(* CODESYS project exsamen m6 no scada.project
   CustomField01_name: CustomField01
   CustomField08_name: CustomField08
   CustomField06_name: CustomField06
   Title: ATV_IMC_Template
   CustomField09_name: CustomField09
   CustomField07_name: CustomField07
   CustomField05_name: CustomField05
   CustomField02_name: CustomField02
   Description: This template can be used for a correct interface with the local drive. the MANDATORY_AT_EACH_CYCLE program must be called like it is done in this application.
   CustomField04_name: CustomField04
   CustomField10_name: CustomField10
   Version: 0.0.0.0
   Company: Schneider Electric
   CustomField03_name: CustomField03

Project tree, tasks and I/O mapping:
  MyController : TM241CE24R, Schneider Electric, order no. TM241CE24R, version 4.0.3.8
    application Application
      task MAST (cyclic, interval 20 ms, priority 15, watchdog 100 ms x 1) calls progprinc
      function HiddenPOU [ST]
      global variables GVL
      program progprinc [SFC]: RojoManual, PlataManual, NegraManual, PlataAuto, NegroAuto, RojoAuto
      function block POU [LD]
      visualisation scada
    DI : Digital Inputs, Schneider Electric, version 4.0.3.8
        input  ibDI_IB1 : BYTE  // IB1
        unmapped channels: IW0
    DQ : Digital Outputs, Schneider Electric, version 4.0.3.8
        output qwDQ_QW0 : WORD  // QW0
        output qbDQ_QB1 : BYTE  // QB1
    Counters : Counters, Schneider Electric, version 4.0.3.8
    Pulse_Generators : Pulse Generators, Schneider Electric, version 4.0.3.8
    Cartridge_1 : Cartridge, Schneider Electric, version 4.0.3.8
    IO_Bus : IO bus - TM3, Schneider Electric, version 4.0.3.8
    COM_Bus : COM bus, Schneider Electric, version 4.0.3.8
    Ethernet_1 : Ethernet Network, Schneider Electric, version 4.0.3.8
    Serial_Line_1 : Serial line, Schneider Electric, version 4.0.3.8
      SoMachine_Network_Manager : SoMachine-Network Manager, Schneider Electric, version 4.0.0.2
    Serial_Line_2 : Serial line, Schneider Electric, version 4.0.3.8
      Modbus_Manager : Modbus Manager, Schneider Electric, version 4.0.0.2
  text list GlobalTextList
*)

// MyController/Application/GVL
VAR_GLOBAL
	Marcha: BOOL;
	Confirmar: BOOL;
	Modo: BOOL;
	
	Bot: INT;
	
	SelecPlata: BOOL;
	SensAlmacenPlata: BOOL;
	SensCilPlata: BOOL;
	
	SelecRojo: BOOL;
	SensAlmacenRojo: BOOL;
	SensCilRojo: BOOL;
	
	SelecNegro: BOOL;
	SensAlmacenNego: BOOL;
	SensCilNegro: BOOL;
	

	Cinta: BOOL;
	Seleccion: BOOL;
END_VAR

// MyController/Application/progprinc
PROGRAM progprinc
VAR
	MarchaPanel: BOOL;
	etapa_0: BOOL;
	etapa_1: BOOL;
	FuncManRojo: POU;
	piezasrojas: INT;
	piezasnegras: INT;
	piezasplata: INT;
	FunManNegra: POU;
	FuncManPlata: POU;
	FuncAutoPlata: POU;
	FuncAutoNegra: POU;
	FuncAutoRoja: POU;

END_VAR

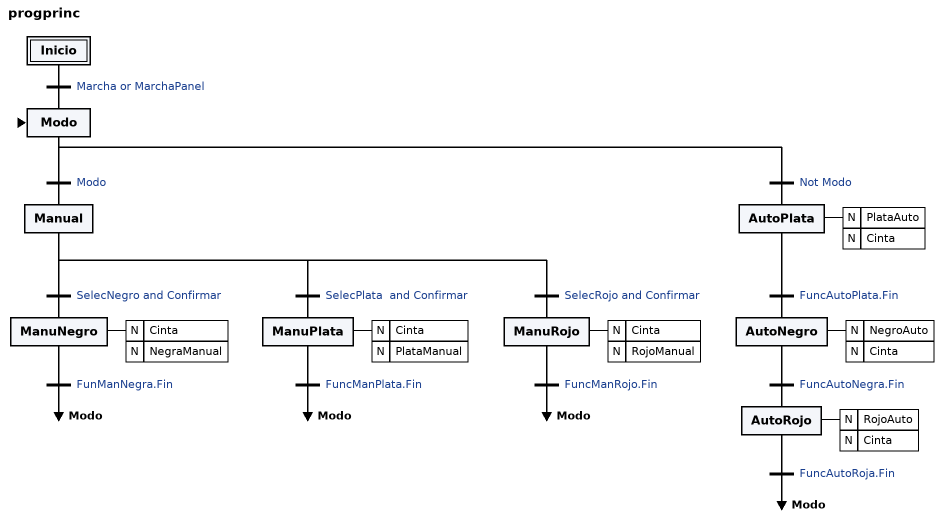
INITIAL_STEP Inicio:
END_STEP
TRANSITION FROM Inicio TO Modo
    := Marcha or MarchaPanel;
END_TRANSITION
STEP Modo:
END_STEP
TRANSITION FROM Modo TO Manual
    := Modo;
END_TRANSITION
STEP Manual:
END_STEP
TRANSITION FROM Manual TO ManuNegro
    := SelecNegro and Confirmar;
END_TRANSITION
STEP ManuNegro:
    Cinta(N);
    NegraManual(N);
END_STEP
TRANSITION FROM ManuNegro TO Modo
    := FunManNegra.Fin;
END_TRANSITION
TRANSITION FROM Manual TO ManuPlata
    := SelecPlata and Confirmar;
END_TRANSITION
STEP ManuPlata:
    Cinta(N);
    PlataManual(N);
END_STEP
TRANSITION FROM ManuPlata TO Modo
    := FuncManPlata.Fin;
END_TRANSITION
TRANSITION FROM Manual TO ManuRojo
    := SelecRojo and Confirmar;
END_TRANSITION
STEP ManuRojo:
    Cinta(N);
    RojoManual(N);
END_STEP
TRANSITION FROM ManuRojo TO Modo
    := FuncManRojo.Fin;
END_TRANSITION
TRANSITION FROM Modo TO AutoPlata
    := Not Modo;
END_TRANSITION
STEP AutoPlata:
    PlataAuto(N);
    Cinta(N);
END_STEP
TRANSITION FROM AutoPlata TO AutoNegro
    := FuncAutoPlata.Fin;
END_TRANSITION
STEP AutoNegro:
    NegroAuto(N);
    Cinta(N);
END_STEP
TRANSITION FROM AutoNegro TO AutoRojo
    := FuncAutoNegra.Fin;
END_TRANSITION
STEP AutoRojo:
    RojoAuto(N);
    Cinta(N);
END_STEP
TRANSITION FROM AutoRojo TO Modo
    := FuncAutoRoja.Fin;
END_TRANSITION

ACTION RojoManual:
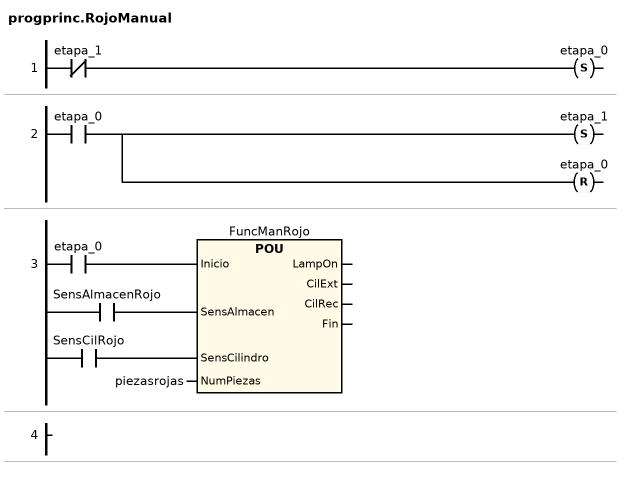
// NETWORK 1
etapa_0 S= NOT etapa_1;

// NETWORK 2
etapa_1 S= etapa_0;
etapa_0 R= etapa_0;

// NETWORK 3
FuncManRojo(
    Inicio := etapa_0,
    SensAlmacen := SensAlmacenRojo,
    SensCilindro := SensCilRojo,
    NumPiezas := piezasrojas); // POU

// NETWORK 4
END_ACTION

ACTION PlataManual:
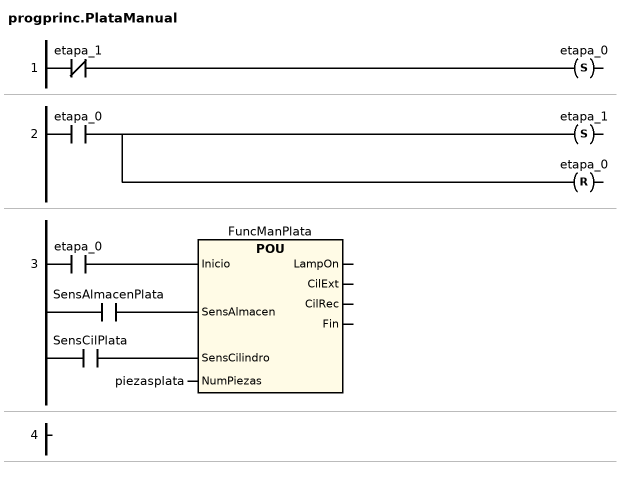
// NETWORK 1
etapa_0 S= NOT etapa_1;

// NETWORK 2
etapa_1 S= etapa_0;
etapa_0 R= etapa_0;

// NETWORK 3
FuncManPlata(
    Inicio := etapa_0,
    SensAlmacen := SensAlmacenPlata,
    SensCilindro := SensCilPlata,
    NumPiezas := piezasplata); // POU

// NETWORK 4
END_ACTION

ACTION NegraManual:
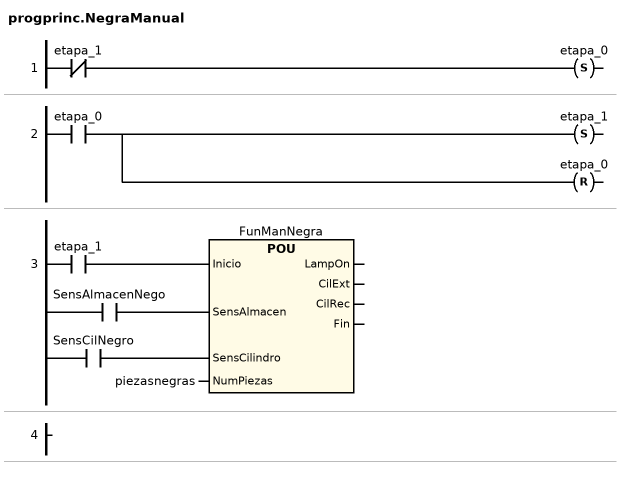
// NETWORK 1
etapa_0 S= NOT etapa_1;

// NETWORK 2
etapa_1 S= etapa_0;
etapa_0 R= etapa_0;

// NETWORK 3
FunManNegra(
    Inicio := etapa_1,
    SensAlmacen := SensAlmacenNego,
    SensCilindro := SensCilNegro,
    NumPiezas := piezasnegras); // POU

// NETWORK 4
END_ACTION

ACTION PlataAuto:
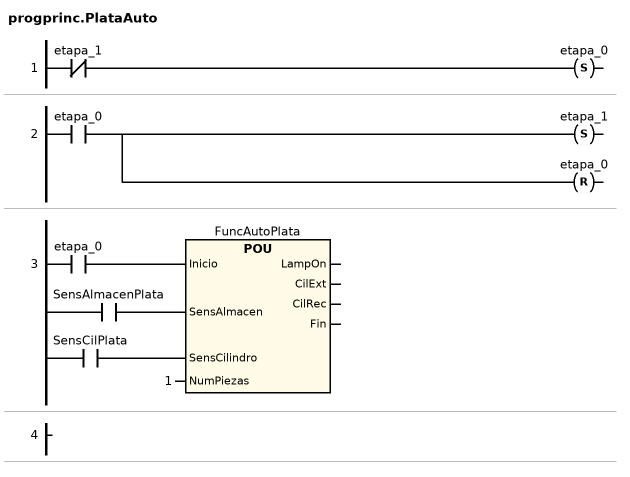
// NETWORK 1
etapa_0 S= NOT etapa_1;

// NETWORK 2
etapa_1 S= etapa_0;
etapa_0 R= etapa_0;

// NETWORK 3
FuncAutoPlata(
    Inicio := etapa_0,
    SensAlmacen := SensAlmacenPlata,
    SensCilindro := SensCilPlata,
    NumPiezas := 1); // POU

// NETWORK 4
END_ACTION

ACTION NegroAuto:
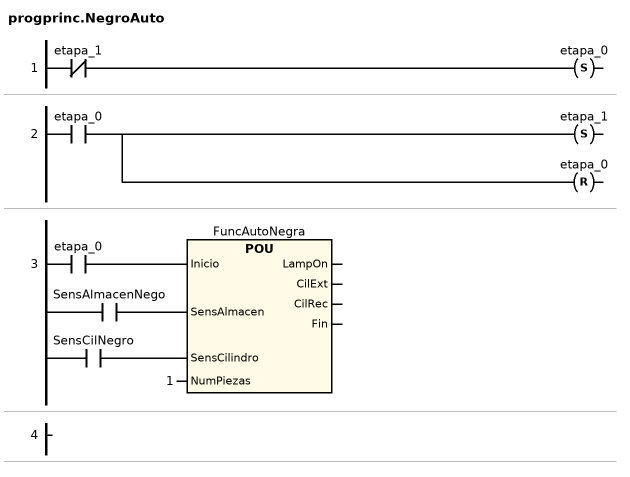
// NETWORK 1
etapa_0 S= NOT etapa_1;

// NETWORK 2
etapa_1 S= etapa_0;
etapa_0 R= etapa_0;

// NETWORK 3
FuncAutoNegra(
    Inicio := etapa_0,
    SensAlmacen := SensAlmacenNego,
    SensCilindro := SensCilNegro,
    NumPiezas := 1); // POU

// NETWORK 4
END_ACTION

ACTION RojoAuto:
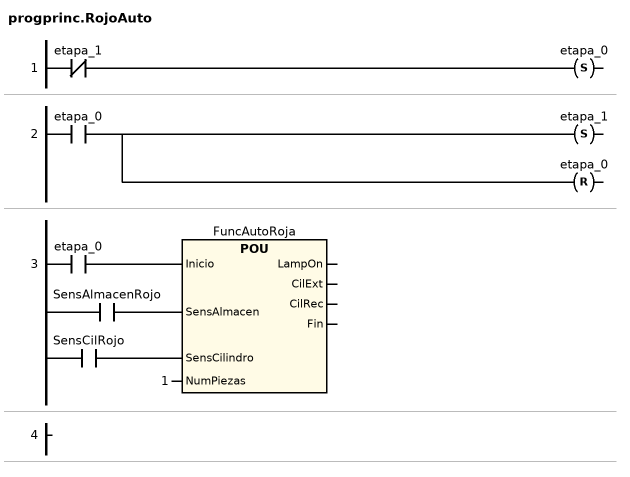
// NETWORK 1
etapa_0 S= NOT etapa_1;

// NETWORK 2
etapa_1 S= etapa_0;
etapa_0 R= etapa_0;

// NETWORK 3
FuncAutoRoja(Inicio := etapa_0, SensAlmacen := SensAlmacenRojo, SensCilindro := SensCilRojo, NumPiezas := 1); // POU

// NETWORK 4
END_ACTION

END_PROGRAM

// MyController/Application/POU
FUNCTION_BLOCK POU

VAR_INPUT
	Inicio: BOOL;
	SensAlmacen: BOOL;
	SensCilindro: BOOL;
	NumPiezas: INT;
END_VAR
VAR_OUTPUT
	CilExt: BOOL;
	CilRec: BOOL;
	LampOn: BOOL;
	Fin: BOOL;
END_VAR
VAR
	etapa_0: BOOL;
	etapa_1: BOOL;
	etapa_2: BOOL;
	etapa_3: BOOL;
	etapa_4: BOOL;
	ContPiezas: BOOL;
	ContadorPiezas: CTU;
	TempSeg: TON;
	
END_VAR
VAR // added by the converter: edge detectors and wires of the graphical bodies
    _w1, _w2, _w3, _w4, _w5 : BOOL;
END_VAR

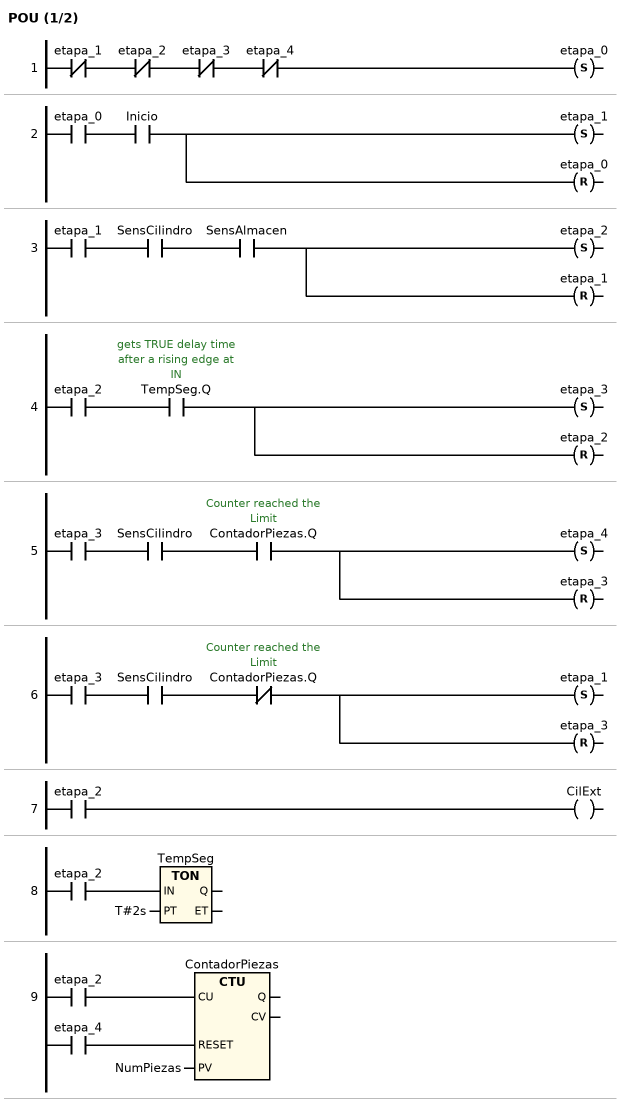
// NETWORK 1
etapa_0 S= NOT etapa_1 AND NOT etapa_2 AND NOT etapa_3 AND NOT etapa_4;

// NETWORK 2
_w1 := etapa_0 AND Inicio;
etapa_1 S= _w1;
etapa_0 R= _w1;

// NETWORK 3
_w2 := etapa_1 AND SensCilindro AND SensAlmacen;
etapa_2 S= _w2;
etapa_1 R= _w2;

// NETWORK 4
//   TempSeg.Q: gets TRUE delay time after a rising edge at IN
_w3 := etapa_2 AND TempSeg.Q;
etapa_3 S= _w3;
etapa_2 R= _w3;

// NETWORK 5
//   ContadorPiezas.Q: Counter reached the Limit
_w4 := etapa_3 AND SensCilindro AND ContadorPiezas.Q;
etapa_4 S= _w4;
etapa_3 R= _w4;

// NETWORK 6
//   ContadorPiezas.Q: Counter reached the Limit
_w5 := etapa_3 AND SensCilindro AND NOT ContadorPiezas.Q;
etapa_1 S= _w5;
etapa_3 R= _w5;

// NETWORK 7
CilExt := etapa_2;

// NETWORK 8
TempSeg(IN := etapa_2, PT := T#2s); // TON

// NETWORK 9
ContadorPiezas(CU := etapa_2, RESET := etapa_4, PV := NumPiezas); // CTU

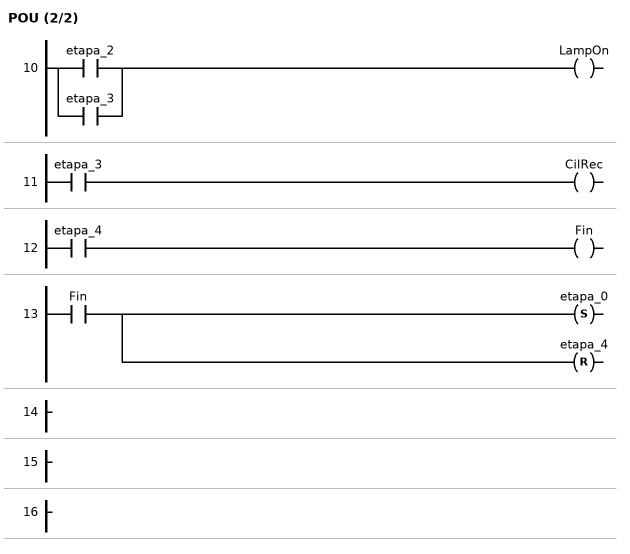
// NETWORK 10
LampOn := etapa_2 OR etapa_3;

// NETWORK 11
CilRec := etapa_3;

// NETWORK 12
Fin := etapa_4;

// NETWORK 13
etapa_0 S= Fin;
etapa_4 R= Fin;

// NETWORK 14

// NETWORK 15

// NETWORK 16

END_FUNCTION_BLOCK

// MyController/Application/HiddenPOU
FUNCTION HiddenPOU : BOOL

VAR_INPUT
	pHiddenFunc: POINTER TO WORD;
END_VAR
VAR
	pRead: POINTER TO BYTE;
	pWrite: POINTER TO BYTE;
END_VAR

pRead := pHiddenFunc + 400;
pWrite := pHiddenFunc + 4400;
HiddenPOU := TRUE;

END_FUNCTION

// MyController/Application/scada
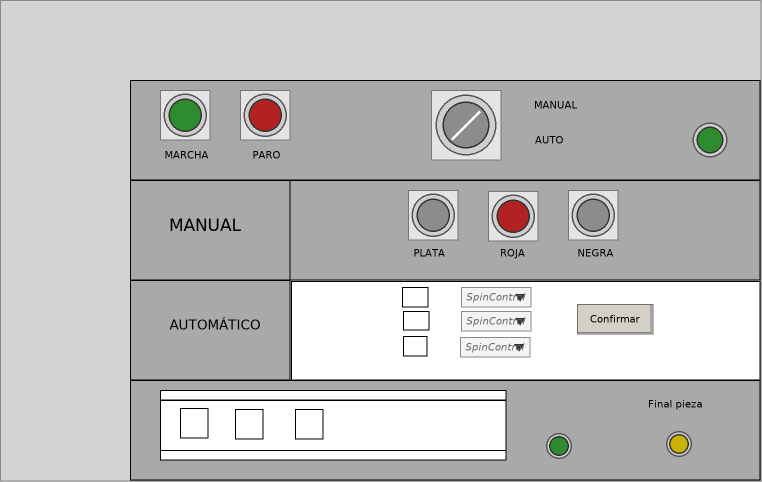
VISUALIZATION scada  // 762x482
    Rectangle (291,281 469x99)
    Rectangle (130,80 630x100)
    Rectangle (130,180 630x100)
    PushSwitch (160,90 50x50), variable: marcha, behaviour: TOGGLE, style: Switch-PushSwitch-Green
    PushSwitch (240,90 50x50), behaviour: TOGGLE, style: Switch-PushSwitch-Red
    Label (150,140 73x30), "MARCHA"
    Label (230,140 73x30), "PARO"
    Lamp1 (690,110 40x60), variable: marcha, style: Lamp-Lamp1-Green
    Rectangle (130,180 160x100)
    Rectangle (130,280 160x100)
    Label (160,210 90x30), "MANUAL"
    Label (150,310 130x30), "AUTOMÁTICO"
    RotarySwitch (431,90 70x70), variable: boton, behaviour: TOGGLE, style: Switch-RotarySwitch-Gray
    Label (519,90 73x30), "MANUAL"
    Label (503,125 93x30), "AUTO"
    Rectangle (130,380 630x100)
    PushSwitch (408,190 50x50), variable: botpla, behaviour: TOGGLE, style: Switch-PushSwitch-Gray
    PushSwitch (568,190 50x50), variable: botnegro, behaviour: TOGGLE, style: Switch-PushSwitch-Gray
    PushSwitch (488,191 50x50), variable: botroj, behaviour: TOGGLE, style: Switch-PushSwitch-Red
    Label (393,238 73x30), "PLATA"
    Label (476,238 73x30), "ROJA"
    Label (559,238 73x30), "NEGRA"
    SpinControl (461,287 70x20)
    SpinControl (461,311 70x20)
    SpinControl (460,337 70x20)
    Button (577,304 76x30), "Confirmar", pressed state: Confirmar
    Rectangle (160,400 346x57)
    Rectangle (160,450 346x10)
    Rectangle (160,390 346x10)
    Lamp1 (664,419 30x50), style: Lamp-Lamp1-Yellow
    Lamp1 (544,421 30x50), style: Lamp-Lamp1-Green
    Label (639,389 73x30), "Final pieza"
    RoundedRectangle (295,409 28x30)
    RoundedRectangle (235,409 28x30)
    RoundedRectangle (180,408 28x30)
    RoundedRectangle (403,336 24x20)
    RoundedRectangle (403,311 26x19)
    RoundedRectangle (402,287 26x20)
END_VISUALIZATION
